(* IEC 61131-3 sources: POMIRTS_lab3/AS/Library_2/MTPATune/V1.00.2, 3 files *)

(* ---- MTPATune.typ ---- *)
TYPE
	MTPATuneFFParametersType : 	STRUCT  (*Finite Frequency Parameters*)
		ControllerType : MTPATuneControllerEnum; (*Type of Controller (PI or PID)*)
		MaxAmplitude : REAL; (*The max value of test signal (applied direct to the plant)*)
		MaxTimeConstant : REAL; (*The biggest plant time constant or plant transient duration*)
		SystemSettlingTime : REAL; (*The desired plant settling time*)
		PhaseMargin : REAL; (*The desired system phase margin*)
		MinOut : REAL; (*Lower manipulated variable limit (lower modulation limit of the subsequent actuator). Permitted range of values: MinOut < MaxOut.*)
		MaxOut : REAL; (*Upper manipulated variable limit (upper modulation limit of the subsequent actuator). Permitted range of values: MaxOut > MinOut.*)
	END_STRUCT;
	MTPATunePIDParametersType : 	STRUCT  (*PID controller Parameters*)
		Gain : REAL; (*Proportional gain. Valid value range: Gain > 0.*)
		IntegrationTime : REAL; (*Integral time constant for the integral component. Unit: [s]. Valid value range: IntegrationTime >= 0.*)
		DerivativeTime : REAL; (*Differential time constant for the derivative component. Unit: [s]. Valid value range: DerivativeTime >= 0.*)
		FilterTime : REAL; (*Filter time constant for the derivative component. Unit: [s]. Valid value range: FilterTime >= 0.*)
		DerivativeGain : REAL; (*Derivative Gain for the derivative component as function of Differential time and Filter time . Unit: [no unit]. Valid value range: FilterTime >= 0.*)
	END_STRUCT;
	MTPATuneFFInternalType : 	STRUCT  (*Data for internal use.*)
		Parameters : MTPATuneFFParametersType; (*Data for internal use.*)
		PIDSelect : BOOL; (*Data for internal use.*)
		RecalculatePIDOld : BOOL; (*Data for internal use.*)
		ParametersValid : BOOL; (*Data for internal use.*)
		Offset : REAL; (*Offset which is used during active tuning procedure.*)
		Error : BOOL; (*Data for internal use.*)
		Warning : BOOL; (*Data for internal use.*)
		UpdateOld : BOOL; (*Data for internal use.*)
		EnableOld : BOOL; (*Data for internal use.*)
		nErrorRegister : UINT; (*Data for internal use.*)
		StartOld : BOOL; (*Data for internal use.*)
		dTuningProgress : REAL; (*Tuning progress in %*)
		dOmegaFilterProgress : REAL; (*Current omega filtering progress in %*)
		dBetaHigh : REAL; (*Data for internal use.*)
		dAlphaHigh : REAL; (*Data for internal use.*)
		dOmegaHigh : REAL; (*Data for internal use.*)
		dBetaLow : REAL; (*Data for internal use.*)
		dAlphaLow : REAL; (*Data for internal use.*)
		dOmegaLow : REAL; (*Data for internal use.*)
		pdBetaPlantOld : ARRAY[0..1]OF REAL; (*Data for internal use.*)
		pdBetaPlant : ARRAY[0..1]OF REAL; (*Data for internal use.*)
		pdAlphaPlantOld : ARRAY[0..1]OF REAL; (*Data for internal use.*)
		pdAlphaPlant : ARRAY[0..1]OF REAL; (*Data for internal use.*)
		pdBetaY : ARRAY[0..1]OF REAL; (*Data for internal use.*)
		pdBetaU : ARRAY[0..1]OF REAL; (*Data for internal use.*)
		pdAlphaY : ARRAY[0..1]OF REAL; (*Data for internal use.*)
		pdAlphaU : ARRAY[0..1]OF REAL; (*Data for internal use.*)
		pdAmpl : ARRAY[0..1]OF REAL; (*Data for internal use.*)
		nArrayCount : USINT; (*Data for internal use.*)
		pdOmegaArray : ARRAY[0..10]OF REAL; (*Data for internal use.*)
		pdBetaArray : ARRAY[0..10]OF REAL; (*Data for internal use.*)
		pdAlphaArray : ARRAY[0..10]OF REAL; (*Data for internal use.*)
		pdOmega : ARRAY[0..1]OF REAL; (*Data for internal use.*)
		dTime : REAL; (*Data for internal use.*)
		timeCURRENT : TIME; (*Data for internal use.*)
		timeINIT : TIME; (*Data for internal use.*)
		dIteration : REAL; (*Data for internal use.*)
		nCalc : BYTE; (*Data for internal use.*)
		nCount : INT; (*Data for internal use.*)
		nPeriodSize : INT; (*Data for internal use.*)
		nPeriodNum : INT; (*Data for internal use.*)
		nPeriodMax : INT; (*Data for internal use.*)
		nPlantOrder : USINT; (*Data for internal use.*)
		dCycleTime : REAL; (*Data for internal use.*)
		byTunerStatus : BYTE; (*Data for internal use.*)
	END_STRUCT;
	MTPATuneControllerEnum :
		( (*Controller Type*)
		mtPAT_PI_Controller := 0, (*PI controller *)
		mtPAT_PID_Controller := 1 (*PID controller*)
		);
END_TYPE

(* ---- MTPATune.fun ---- *)
{REDUND_OK} FUNCTION_BLOCK MTPATuneFiniteFrequency (*Parametric dynamic model indentification combined with loop shaping based PID tuning*)
	VAR_INPUT
		Enable : BOOL; (*Enables/Disables the function block.*)
		Parameters : MTPATuneFFParametersType; (*Function block parameters.*)
		Update : BOOL; (*Updates the parameters listed above on a rising edge.*)
		Offset : REAL; (*Offset which is added to output Out. Offset kept constant during active tuning procedure.*)
		Start : BOOL; (*Starts the tuning on rising edge.*)
		PlantInput : REAL; (*Current plant input signal.*)
		PlantOutput : REAL; (*Current plant output signal.*)
		RecalculateController : BOOL; (*Calculates the controller parameters again without identification on a rising edge (onle if tuning was carried out once).*)
	END_VAR
	VAR_OUTPUT
		Active : BOOL; (*Function block is active.*)
		Error : BOOL; (*Indicates an error.*)
		StatusID : DINT; (*Status information.*)
		UpdateDone : BOOL; (*Update is done.*)
		TuningActive : BOOL; (*Tuning is active.*)
		TuningDone : BOOL; (*Tuning completed.*)
		Out : REAL; (*Output value (manipulated variable).*)
		PIDParameters : MTPATunePIDParametersType; (*PID parameters.*)
		Numerator : ARRAY[0..1] OF REAL; (*Coefficients of plant transer function nominator: k(s) = b[1]*s +  b[0]*) (* *) (*#PAR#*)
		Denominator : ARRAY[0..2] OF REAL; (*Coefficients of plant transer function denominator: d(s) =a[2] * s^2 +  a[1] * s + a[0]*) (* *) (*#PAR#*)
	END_VAR
	VAR
		Internal : MTPATuneFFInternalType; (*Data for internal use.*)
	END_VAR
END_FUNCTION_BLOCK

(* ---- MTPATune.var ---- *)
(*Error*)
VAR CONSTANT
	mtPAT_ERR_SMALL_MAX_TIME_CONST : DINT := -1058004075; (*In test signal the frequency is so high that its period is less than 20 sampling time. Tuning results are not issued when this error. The procedure should be restart with MaxTimeConstant increased.*)
	mtPAT_ERR_PID_TUNING_FAILED : DINT := -1058004074; (*The unstable model is identified from measured data. Tuning results are not issued when this error.*)
	mtPAT_ERR_INVALID_PLANT_IO : DINT := -1058004073; (*"PlantInput" and or "PlantOutput" loaded with NAN or +-Inf*)
	mtPAT_ERR_INVALID_MAX_TIME_CONST : DINT := -1058004072; (*Invalid Parameter "MaxTimeConstant"*)
	mtPAT_ERR_INVALID_MAX_AMPLITUDE : DINT := -1058004071; (*Invalid Parameter "MaxAmplitude"*)
	mtPAT_ERR_INVALID_PHASE_MARGIN : DINT := -1058004070; (*Invalid Parameter "PhaseMargin". Either "PhaseMargin" = 0 or "PhaseMargin">=45° and "PhaseMargin"<=90°*)
	mtPAT_ERR_INVALID_OUT_LIMITATION : DINT := -1058004069; (*Invalid Parameter "MinOut" and / or MaxOut. Either "MinOut" = "MaxOut" = 0 or "MinOut" < "MaxOut".*)
	mtPAT_ERR_OUTPUT_SATURATION : DINT := -1058004068; (*Tuning was aborted because output "Out" was limited by "MinOut" or "MaxOut".*)
	mtPAT_ERR_PID_RECALC_FAILED : DINT := -1058004067; (*Procedure of PID controller parameters recalculation (fbTuner.bPID_Recalc is true) can not be executed because there is no the model data or fbTuner.bFinish is false.*)
END_VAR
(*Warning*)
VAR CONSTANT
	mtPAT_WRN_INVALID_IDENT_VERIFY : DINT := -2131745900; (* Verification of identification results is mismatched. This is a warning. Results are present but may be incorrect.*)
	mtPAT_WRN_NO_TUNING_CONVERGENCE : DINT := -2131745899; (*This is a warning that within stated identification time the convergence condition is not satisfied.  Results are present but may be incorrect. *)
	mtPAT_WRN_MAX_IT_LOW_FREQ_SEARCH : DINT := -2131745898; (*Procedure of low-frequency search exceeds a predetermined number of iterations. This is a warning that the procedure is not followed through. Most likely it does not affect the quality of the result or the procedure should be restart with MaxTimeConstant increased.*)
	mtPAT_WRN_INVALID_MAX_TIME_CONST : DINT := -2131745897; (*Invalid Parameter "MaxTimeConstant"*)
	mtPAT_WRN_INVALID_MAX_AMPLITUDE : DINT := -2131745896; (*Invalid Parameter "MaxAmplitude"*)
	mtPAT_WRN_INVALID_PHASE_MARGIN : DINT := -2131745895; (*Invalid Parameter "PhaseMargin". Either "PhaseMargin" = 0 or "PhaseMargin">=45° and "PhaseMargin"<=90°.*)
	mtPAT_WRN_INVALID_OUT_LIMITATION : DINT := -2131745894; (*Invalid Parameter "MinOut" and / or MaxOut. Either "MinOut" = "MaxOut" = 0 or "MinOut" < "MaxOut".*)
	mtPAT_WRN_PID_CALC_MAX_ITER : DINT := -2131745893; (*Procedure of calculation of PID controller parameters exceeds a predetermined number of iterations. This is a warning that actual phase margin is less than Parameter "PhaseMargin" and controller is not robust. Problem can be solved by increasing of the value of SystemSettlingTime.*)
END_VAR
